// TIA Portal V19 export
DATA_BLOCK "DB_PNOZ_IN_Out"   // DB361
TITLE = DB99 V0.4
{ S7_Optimized_Access := 'FALSE' }
AUTHOR : MW_CSTS
FAMILY : PNOZmc_p
VERSION : 0.4
// für PNOZmulti m1p ab V5.6
// stored: AutoNumber false
   VAR
      In : Struct
         Header : Array[0..7] of Byte;
         PNOZ_OK : Bool := false;   // kein NotHalt global aktiv
         "NH-T_SS_ok" : Bool;   // NH-Taster Schaltschrank o.k.
         "NH-T_Filter_ok" : Bool;   // NH-Taster Filterstation o.k.
         "NH-T_Vers_ok" : Bool;   // NH-Taster Versorgung o.k.
         "NH-T_Ents_ok" : Bool;   // NH-Taster Entsorgung o.k.
         "NH-T_Vent_ok" : Bool;   // NH-Taster Ventilator o.k.
         NH_Koppl_ok : Bool;   // NH Koppl. Res. o.k.
         NH_MP_ok : Bool;   // NH Mobile Panel o.k.
         Tuer_VS_ok : Bool := false;   // Tür Vorderseite o.k.
         Tuer_RS_ok : Bool;   // Tür Rückseite o.k.
         "SRM_Zu_BG-QM43" : Bool;   // SRM ZU UV GP02.BG-QM43
         "SRM_Auf_BG-QM43" : Bool;   // SRM AUF UV GP02.BG-QM43
         "SRM_Zu_BG-QM44" : Bool;   // SRM ZU UV GP02.BG-QM44
         "SRM_Auf_BG-QM44" : Bool;   // SRM AUF UV GP02.BG-QM44
         Abluft_ok : Bool;   // Abluft o.k.
         Tuer_zu_Seite_GP01 : Bool := false;   // Tür geschlossen Seite GP01
         Tuer_zu_vorn_GP01 : Bool := false;   // Tür geschlossen vorn GP01
         Tuer_zu_vorn_GP02 : Bool := false;   // Tür geschlossen vorn GP02
         FG_zu_HQ01 : Bool := false;   // Filtereinhausung geschloosen HQ01.BG06
         FG_zu_HQ02 : Bool := false;   // Filtereinhausung geschloosen HQ02.BG09
         T_Aktion_MP : Bool := false;   // Aktionstaster MobilePanel
         NH_Frg_TW_QF : Bool := false;   // Freigabe Nothalt Transportsystem
         NH_Frg_Pumpen : Bool := false;   // Freigabe Nothalt Pumpen
         NH_Frg_FP_CM01 : Bool := false;   // Freigabe Nothalt Filterpumpe CM01
         NH_Frg_FP_CM02 : Bool := false;   // Freigabe Nothalt Filterpumpe CM02
         NH_Frg_Deckel : Bool := false;   // Freigabe Not-Halt Deckel
         NH_Frg_RT : Bool := false;   // Freigabe Not-Halt Rolltor
         "res11.3" : Bool;
         "res11.4" : Bool;
         "res11.5" : Bool;
         "res11.6" : Bool;
         "res11.7" : Bool;
         VirtualInput : Array[32..127] of Bool;
         LED_0_Fault : Bool;   // LED 0 Fault
         LED_1_Fault : Bool;   // LED 1 Fault
         LED_Fault : Bool;   // LED Fault
         LED_Diag : Bool;   // LED Diag
         LED_Run_ST : Bool := false;   // LED Run ST
         reserved1 : Bool;   // reserved
         LED_Run_FS : Bool := false;   // LED Run FS
         Data_cons_check_bit : Bool;   // Data consistence check bit
         Table_Nr : Byte;   // Table Nr
         Segment : Struct
            Nr : Byte;
            Byte_0 : Byte;
            Byte_1 : Byte;
            Byte_2 : Byte;
            Byte_3 : Byte;
            Byte_4 : Byte;
            Byte_5 : Byte;
            Byte_6 : Byte;
            Byte_7 : Byte;
            Byte_8 : Byte;
            Byte_9 : Byte;
            Byte_10 : Byte;
            Byte_11 : Byte;
            Byte_12 : Byte;
         END_STRUCT;
         reserviert : Byte;
         Checksum : Byte := BYTE#16#0;   // Checksumme, Byte 4 + Byte 39
         Endekennung : Byte := BYTE#16#10;   // last Byte, must be 0x10 every time!
         Struct_Auffueller : Byte;
      END_STRUCT;
      Out : Struct
         Header : Array[0..7] of Byte;
         T_NH_Quitt : Bool;   // Taster Not-Halt Quittierung
         Frg_Automatik : Bool;   // Freigabe Automatik Transportsystem
         res_2 : Bool;
         res_3 : Bool;
         res_4 : Bool;
         res_5 : Bool;
         res_6 : Bool;
         res_7 : Bool;
         res_8 : Bool;
         res_9 : Bool;
         res_10 : Bool;
         res_11 : Bool;
         res_12 : Bool;
         res_13 : Bool;
         res_14 : Bool;
         res_15 : Bool;
         VirtualOutput : Array[16..127] of Bool;
         LED : Byte;
         Req_Table_Nr : Byte;   // Table Nr
         Segment : Struct
            Req_Nr : Byte;
            Byte_0 : Byte;
            Byte_1 : Byte;
            Byte_2 : Byte;
            Byte_3 : Byte;
            Byte_4 : Byte;
            Byte_5 : Byte;
            Byte_6 : Byte;
            Byte_7 : Byte;
            Byte_8 : Byte;
            Byte_9 : Byte;
            Byte_10 : Byte;
            Byte_11 : Byte;
            Byte_12 : Byte;
         END_STRUCT;
         reserviert : Byte;
         Checksum : Byte := BYTE#16#A4;   // Checksumme, Byte 4 + Byte 39
         Endekennung : Byte := BYTE#16#10;   // last Byte, must be 0x10 every time!
         Struct_Auffueller : Byte;
      END_STRUCT;
   END_VAR
BEGIN
   In.Header[0] := BYTE#16#05;
   In.Header[1] := BYTE#16#15;
   In.Header[3] := BYTE#16#26;
   In.Header[4] := BYTE#16#DC;
   Out.Header[0] := BYTE#16#05;
   Out.Header[1] := BYTE#16#15;
   Out.Header[3] := BYTE#16#26;
   Out.Header[4] := BYTE#16#5C;
END_DATA_BLOCK
